(* IEC 61131-3 sources: SigmatekTestframework/src/Class/CJUnitReport, 1 file *)

(* ---- CJUnitReport.st ---- *)
#define XML_VERSION     "<?xml version=$221.0$22 encoding=$22UTF-8$22?>"
#define XML_TESTSUITE   "$t<testsuite name=$22%1$22 tests=$22%2$22 disabled=$22%3$22 failures=$22%5$22>"
#define XML_TESTCASE    "$t$t<testcase name=$22%1$22 assertions=$22%2$22 classname=$22%3$22 time=$22%4$22 package=$22%5$22>"
#define XML_TESTPASSED  "$t$t$t<passed/>$n"
#define XML_TESTSKIPPED "$t$t$t<skipped/>$n"
#define XML_TESTFAILED  "$t$t$t<failure message=$22%1$22/>$n"

(*!
<Class
	Name               = "CJUnitReport"
	Revision           = "1.0"
	RealtimeTask       = "false"
	CyclicTask         = "false"
	BackgroundTask     = "false"
	Sigmatek           = "false"
	OSInterface        = "false"
	HighPriority       = "false"
	Automatic          = "false"
	UpdateMode         = "Prescan"
	SharedCommandTable = "true"
	Objectsize         = "(510,120)">
	<Channels>
	</Channels>
	<Network Name="CJUnitReport">
		<!-- List of Components in this network -->
		<Components>
			<Object
				Name       = "_base"
				Class      = "CTestReportBase"
				Position   = "(218,120)"
				Visualized = "false">
				<Channels>
					<Server Name="Registered"/>
					<Client Name="clib"/>
					<Client Name="File"/>
					<Client Name="System"/>
				</Channels>
			</Object>
		</Components>
		<Comments>
		</Comments>
		<!-- List of Connections in this network -->
		<Connections>
			<Connection Source="this.Registered" Destination="_base.Registered" Vertices="(690,210),(518,210),"/>
			<Connection Source="_base.File" Destination="this.File" Vertices="(218,210),(38,210),"/>
		</Connections>
		<!-- Headerfiles -->
		<Options>
		</Options>
	</Network>
</Class>
*)
#pragma using CTestReportBase

CJUnitReport : CLASS
: CTestReportBase
	TYPE
	  EExport_t :
	  (
	    eInit,
	    eExportTestSuite,
	    eExportTestcase,
	    eNextTestSuite,
	    eFinish
	  )$UDINT;
	END_TYPE
  //Servers:
  //Clients:
  //Variables:
		m_itSuite 	: CLinkedList::Iterator_t;
		m_itCase 	: CLinkedList::Iterator_t;
		eExportState 	: EExport_t;
		pTestSuite 	: ^CTestSuite;
		pTestcase 	: ^CTestBase;
  //Functions:

	FUNCTION VIRTUAL BuildFile
		VAR_OUTPUT
			eRetcode 	: ERetCode_t;
		END_VAR;

	FUNCTION VIRTUAL getFileName
		VAR_INPUT
			pFileName 	: ^CHAR;
			pFilePath 	: ^CHAR;
		END_VAR
		VAR_OUTPUT
			eRetcode 	: ERetCode_t;
		END_VAR;
  //Tables:
	FUNCTION @STD
		VAR_OUTPUT
			ret_code	: CONFSTATES;
		END_VAR;
	FUNCTION GLOBAL TAB @CT_;
END_CLASS;

#pragma usingLtd CTestBase
#pragma usingLtd CTestSuite

//Exclude-SccX
(*
 **********************************************************************
 * \file CXmlTestReport.st
 *
 * Creates a simple XML-File as report
 *
 * Copyright (c) 2016,Hoox.Software, Helmbrechts
 * All Rights Reserved.
 *
 * Created on: 01.06.2016
 *     Author: dressel
 *
 **********************************************************************
 *)
#pragma using CTestSuite
#pragma using CTestBase
//*********************************************************************
//
//
//
//
//*********************************************************************
FUNCTION VIRTUAL CJUnitReport::getFileName
	VAR_INPUT
		pFileName 	: ^CHAR;
		pFilePath 	: ^CHAR;
	END_VAR
	VAR_OUTPUT
		eRetcode 	: ERetCode_t;
	END_VAR

   _strcpy(dest:= pFilePath, src:= "C:\testrun");
   _strcpy(dest:= pFileName, src:= "junit.xml");

   eRetcode := eDone;

END_FUNCTION

//*********************************************************************
//
//
//
//
//*********************************************************************
FUNCTION VIRTUAL CJUnitReport::BuildFile
	VAR_OUTPUT
		eRetcode 	: ERetCode_t;
	END_VAR
   VAR
      eTestState : CTestBase::ETestState_t;
      buffer     : CTestBase::ABuffer_t;
   END_VAR

   eRetcode := eBusy;

   _memset(dest:=#buffer[0], usByte:=0, cntr:=sizeof(buffer));

   case eExportState of

   eInit:

      clearBuffer();

      addString(XML_VERSION);
      writeBuffer();

      // <Created Date=dd.mm.yy Time=hh.mm.ss>
      addString("<?Created Date=$22");
      addDate(#m_sSysDate);
      addString("$22 Time=$22");
      addTime(#m_sSysTime);
      addString("$22 ?>");
      writeBuffer();

      addString("<testsuites>");
      writeBuffer();

      m_itSuite := m_pTestLib^.getFirstTestsuite();

      if m_itSuite > 0 then
         eExportState := eExportTestSuite;
      else
         eExportState := eFinish;
      end_if;

   eExportTestSuite:

      pTestSuite := m_pTestLib^.getElement(m_itSuite);

      addString(XML_TESTSUITE);

      pTestSuite^.getName(#buffer);
      replace(nil, pReplace:="%1", pData:= #buffer[0]);

      pTestSuite^.getCount(#buffer, CTestsuite::eAll);
      replace(nil, pReplace:="%2", pData:= #buffer[0]);

      pTestSuite^.getCount(#buffer, CTestsuite::eSkipped);
      replace(nil, pReplace:="%3", pData:=#buffer[0]);

      pTestSuite^.getCount(#buffer, CTestsuite::eFailed);
      replace(nil, pReplace:="%5", pData:=#buffer[0]);

      replace(nil, pReplace:="%6", pData:= "Localhost");
      writeBuffer();

      m_itCase := pTestSuite^.getFirstTestcase();

      if m_itCase > 0 then
         eExportState := eExportTestcase;
      end_if;

   eExportTestcase:

      pTestcase := pTestSuite^.getElement(m_itCase);

      // kompletter Eintrag pro Testfall
      //"$t$t<testcase name=$22$22 assertions=$22$22 classname=$22$22 time=$22$22 package=$22$22>"
      addString(XML_TESTCASE);
      pTestCase^.getTestId(#buffer);
      replace(nil, pReplace:="%1", pData:= #buffer[0]);
      pTestCase^.getAsserts(#buffer);
      replace(nil, pReplace:="%2", pData:= #buffer[0]);
      pTestCase^.getFullPath(#buffer);
      replace(#buffer[0], pReplace:="/", pData:= ".");
      replace(nil, pReplace:="%3", pData:= #buffer[0]);
      pTestCase^.getTime(#buffer);
      replace(nil, pReplace:="%4", pData:= #buffer[0]);
      pTestCase^.getPackage(#buffer);
      replace(#buffer[0], pReplace:="/", pData:= ".");
      replace(nil, pReplace:="%5", pData:= #buffer[0]);
      writeBuffer();

      eTestState := ETestState_t::eStateSkipped;
      if pTestSuite^.isSelected() then
         eTestState := pTestCase^.getTestState();
      end_if;

      case eTestState of

      ETestState_t::eStatePassed:

         addString(XML_TESTPASSED);

      ETestState_t::eStateSkipped:

         addString(XML_TESTSKIPPED);

      ETestState_t::eStateFailed:

         addString(XML_TESTFAILED);
         pTestCase^.getMessage(#buffer);
         replace(nil, pReplace:="%1", pData:= #buffer[0]);

      end_case;

      addString("$t$t</testcase>");
      writeBuffer();

      m_itCase := pTestSuite^.getNextTestcase(m_itCase);

      if m_itCase = 0 then
         eExportState := eNextTestSuite;
      end_if;

   eNextTestSuite:

      m_itSuite := m_pTestLib^.getNextTestSuite(m_itSuite);
      addString("$t</testsuite>");
      writeBuffer();

      if m_itSuite > 0 then
         eExportState := eExportTestSuite;
      else
         eExportState := eFinish;
      end_if;

   eFinish:

      addString("</testsuites>");
      writeBuffer();
      eExportState := eInit;
      eRetcode := eDone;

   end_case;

END_FUNCTION
